(* IEC 61131-3 sources: AXOpen/src/showcase/app/src/core/AXOpen.Dialogs, 3 files *)

(* ---- AxoAlertDocuExample.st ---- *)
USING AXOpen.Core;

NAMESPACE AxoAlertExamples

    {S7.extern=ReadWrite}
    CLASS AxoAlertDocuExample EXTENDS AXOpen.Core.AxoObject
        //<AlertDeclaration>
        VAR PUBLIC
            {#ix-set:AttributeName = "<#Process Alert#>"}
            _alert : AXOpen.Core.AxoAlert;
        END_VAR
        //</AlertDeclaration>

        //<AlertUsageVariables>
        VAR PUBLIC
            {#ix-set:AttributeName = "<#Trigger alert#>"}
            _triggerAlert : BOOL;
            {#ix-set:AttributeName = "<#Alert was shown#>"}
            _alertWasShown : BOOL;
        END_VAR
        //</AlertUsageVariables>

        METHOD PUBLIC Execute
            //<AlertShowPattern>
            // AxoAlert shows a timed notification banner on the HMI.
            // Unlike AxoDialog, it does NOT wait for user response.
            // IsShown() returns TRUE once the alert has been displayed and dismissed.
            IF _triggerAlert THEN
                IF _alert.Show(THIS)
                    .WithTitle('<#Process Notification#>')
                    .WithType(eDialogType#Info)
                    .WithMessage('<#Cycle completed successfully.#>')
                    .WithTimeToBurn(UINT#5).IsShown() THEN
                    // Alert was displayed and timed out
                    _alertWasShown := TRUE;
                    _triggerAlert := FALSE;
                END_IF;
            END_IF;
            //</AlertShowPattern>
        END_METHOD

        METHOD AlertTypeExamples
        //<AlertTypes>
            // Info alert — general information
            IF _alert.Show(THIS)
                .WithTitle('<#Info#>')
                .WithType(eDialogType#Info)
                .WithMessage('<#Operation started.#>')
                .WithTimeToBurn(UINT#3).IsShown() THEN
                ;
            END_IF;

            // Success alert — operation completed
            IF _alert.Show(THIS)
                .WithTitle('<#Success#>')
                .WithType(eDialogType#Success)
                .WithMessage('<#Part inspection passed.#>')
                .WithTimeToBurn(UINT#5).IsShown() THEN
                ;
            END_IF;

            // Warning alert — attention needed
            IF _alert.Show(THIS)
                .WithTitle('<#Warning#>')
                .WithType(eDialogType#Warning)
                .WithMessage('<#Approaching maintenance interval.#>')
                .WithTimeToBurn(UINT#8).IsShown() THEN
                ;
            END_IF;

            // Danger alert — critical condition
            IF _alert.Show(THIS)
                .WithTitle('<#Danger#>')
                .WithType(eDialogType#Danger)
                .WithMessage('<#Emergency stop triggered.#>')
                .WithTimeToBurn(UINT#10).IsShown() THEN
                ;
            END_IF;
        //</AlertTypes>

        //<AlertRestore>
            // Restore clears the alert state, allowing it to be shown again
            _alert.Restore();
        //</AlertRestore>
        END_METHOD
    END_CLASS
END_NAMESPACE

(* ---- AxoDialogExamples.st ---- *)
USING AXOpen.Core;

NAMESPACE AxoDialogExamples

    {S7.extern=ReadWrite}
    CLASS Dialogs EXTENDS AXOpen.Core.AxoObject
        //<DialogDeclaration>
        VAR PUBLIC

            {#ix-set:AttributeName = "Restore All"}
            _invokeRestoreAll : BOOL;

            {#ix-set:AttributeName = "Call ALL"}
            _invokeCallAll : BOOL;

            {#ix-set:AttributeName = "Call ALL in Sequnce"}
            _invokeSequnceAll : BOOL;

             {#ix-set:AttributeName = "Dialog AA"}
             AA : AxoDialogTest;

             {#ix-set:AttributeName = "Dialog BB"}
             BB : AxoDialogTest;

             init_done : bool := false;
        END_VAR
        //</DialogDeclaration>
        VAR PRIVATE
            _rootObject : AxoObject;
        END_VAR

        METHOD PUBLIC Execute
            //<DialogExecution>
            if not init_done THEN
                AA.Caption := 'AA caption';
                BB.Caption := 'BB caption';

                AA.Question := 'AA Question';
                BB.Question := 'BB Question';

                init_done := true;
            end_if;

            IF _invokeRestoreAll THEN
                AA._restoreDialog := TRUE;
                BB._restoreDialog := TRUE;
                _invokeRestoreAll := FALSE;
            END_IF;

            IF _invokeCallAll THEN
                AA._callDialog := TRUE;
                BB._callDialog := TRUE;
                _invokeCallAll := FALSE;
            END_IF;

            IF _invokeSequnceAll THEN
                AA._callDialogInSequnce := TRUE;
                BB._callDialogInSequnce := TRUE;
                _invokeSequnceAll := FALSE;
            END_IF;

            _rootObject.Run(THIS);
            AA.Run(_rootObject);
            BB.Run(_rootObject);
            //</DialogExecution>
        END_METHOD
    END_CLASS
END_NAMESPACE

(* ---- AxoDialogTest.st ---- *)
USING AXOpen.Core;

NAMESPACE AxoDialogExamples

    {S7.extern=ReadWrite}
    CLASS AxoDialogTest EXTENDS AxoObject
        VAR PUBLIC

            {#ix-set:AttributeName = "Restore dialog"}
            _restoreDialog : BOOL;

            {#ix-set:AttributeName = "Call dialog"}
            _callDialog : BOOL;

            {#ix-set:AttributeName = "Call dialog in sequnce"}
            _callDialogInSequnce : BOOL;
            {#ix-set:AttributeName = "Iteration"}
            _iterationStep : INT;
            _timeOutCounter : INT;

            {#ix-set:AttributeName = "Generate Alerts in sequnce"}
            _alertInSequnce : BOOL;
            _alertIterationStep : INT;

            {#ix-set:AttributeName = "External Button signal - OK"}
            _externButtonSignal_ok : BOOL;
            {#ix-set:AttributeName = "External Button signal - YES"}
            _externButtonSignal_yes : BOOL;
            {#ix-set:AttributeName = "External Button signal - NO"}
            _externButtonSignal_no : BOOL;
            {#ix-set:AttributeName = "External Button signal - CANCEL"}
            _externButtonSignal_cancel : BOOL;

            Caption : STRING := 'Caption';
            Question : STRING := 'Question';

            {#ix-set:AttributeName = "Dialog Answer"}
            _answer : eDialogAnswer;

            {#ix-set:AttributeName = "Dialog"}
            _dialog : AXOpen.Core.AxoDialog;

            {#ix-set:AttributeName = "Alert Dialog"}
            _alertDialog : AXOpen.Core.AxoAlert;
        END_VAR

        METHOD PUBLIC OVERRIDE Run
            VAR_INPUT
                inParent : IAxoObject;
            END_VAR;

            SUPER.Run(inParent);
            // THIS.InitializeWithContext(_context);

            IF(_restoreDialog) THEN
                _restoreDialog := false;
                _dialog.Restore();
                _alertDialog.Restore();
                _callDialog:= false;
                _callDialogInSequnce := false;
                _iterationStep := 0;
                _timeOutCounter := 0;

                _alertInSequnce := FALSE;
                _alertIterationStep := 0;
            END_IF;

            //<DialogShowSimplePattern>
            //----------------------  SIMPLE DIALOG (HMI-only response) -------
            IF(_callDialog) THEN
               _answer := _dialog.Show(THIS)
                                  .WithCaption(Caption)
                                  .WithText(Question)
                                  .WithYesNoCancel()
                                  .WithType(eDialogType#Warning)
                                  .Answer();

                IF _answer <> eDialogAnswer#NoAnswer THEN
                    _callDialog := FALSE;
                END_IF;
            END_IF;
            //</DialogShowSimplePattern>

            //<DialogShowWithExternalClosePattern>
            //----------------------  DIALOG WITH EXTERNAL CLOSE SIGNALS -------
            IF(_callDialog) THEN
               _answer := _dialog.ShowWithExternalClose(THIS, _externButtonSignal_ok, _externButtonSignal_yes, _externButtonSignal_no, _externButtonSignal_cancel)
                                                .WithYesNoCancel()
                                                .WithType(eDialogType#Warning)
                                                .WithCaption(Caption)
                                                .WithText(Question)
                                                .Answer();

                IF _answer <> eDialogAnswer#NoAnswer THEN
                    _callDialog := FALSE;
                END_IF;
            END_IF;
            //</DialogShowWithExternalClosePattern>

            //<DialogSequencePattern>
            //----------------------  DIALOG IN SEQUNCE-------------------
            IF _callDialogInSequnce THEN

                if  _iterationStep  = 0 then
                    _iterationStep := _iterationStep + 1;
                end_if;

                if  _iterationStep  = 1 then

                    if not _dialog.HasError() then
                        _answer := _dialog.ShowWithExternalClose(THIS, _externButtonSignal_ok, _externButtonSignal_yes, _externButtonSignal_no, _externButtonSignal_cancel)
                        .WithYesNoCancel()
                        .WithType(eDialogType#Info)
                        .WithCaption( 'Iteraion 1')
                        .WithText(Question)
                        .Answer();

                        THIS.Watcher_Monitor();
                        if _answer <> eDialogAnswer#NoAnswer THEN
                            THIS.Watcher_Reset();
                            _iterationStep := _iterationStep + 1;
                        END_IF;

                    end_if;

                end_if;

                if  _iterationStep  = 2 then

                    if not _dialog.HasError() then
                        _answer := _dialog.ShowWithExternalClose(THIS, _externButtonSignal_ok, _externButtonSignal_yes, _externButtonSignal_no, _externButtonSignal_cancel)
                        .WithYesNoCancel()
                        .WithType(eDialogType#Success)
                        .WithCaption('Iteraion 2')
                        .WithText(Question)
                        .Answer();

                        THIS.Watcher_Monitor();
                        if _answer <> eDialogAnswer#NoAnswer THEN
                            THIS.Watcher_Reset();
                            _iterationStep := _iterationStep + 1;
                        END_IF;
                    end_if;

                end_if;

                if  _iterationStep  = 3 then
                    if not _dialog.HasError() then
                        _answer := _dialog.ShowWithExternalClose(THIS, _externButtonSignal_ok, _externButtonSignal_yes, _externButtonSignal_no, _externButtonSignal_cancel)
                        .WithYesNoCancel()
                        .WithType(eDialogType#Warning)
                        .WithCaption('Iteraion 3')
                        .WithText(Question)
                        .Answer();

                        THIS.Watcher_Monitor();
                        if _answer <> eDialogAnswer#NoAnswer THEN
                            THIS.Watcher_Reset();
                            _iterationStep := _iterationStep + 1;
                        END_IF;
                    end_if;

                end_if;

                if  _iterationStep  = 4 then
                    if not _dialog.HasError() then
                        _answer := _dialog.ShowWithExternalClose(THIS, _externButtonSignal_ok, _externButtonSignal_yes, _externButtonSignal_no, _externButtonSignal_cancel)
                        .WithYesNoCancel()
                        .WithType(eDialogType#Danger)
                        .WithCaption('Iteraion 4')
                        .WithText(Question)
                        .Answer();

                        THIS.Watcher_Monitor();
                        if _answer <> eDialogAnswer#NoAnswer THEN
                            THIS.Watcher_Reset();
                            _iterationStep := _iterationStep + 1;
                        END_IF;
                    end_if;

                end_if;

            end_if;
            //</DialogSequencePattern>
            //<AlertDialogPattern>
            //---------------------- ALERT DIALOG -------------------
            IF _alertInSequnce THEN

                if  _alertIterationStep  = 0 then
                    _alertIterationStep := _alertIterationStep + 1;
                end_if;

                if  _alertIterationStep  = 1 then
                    if not _alertDialog.HasError() then
                        IF _alertDialog.Show(THIS)
                            .WithTitle(Caption)
                            .WithType(eDialogType#Info)
                            .WithMessage('Alert stage 1!')
                            .WithTimeToBurn(UINT#5).IsShown()  THEN
                            //when task is done, move next
                            _alertIterationStep := _alertIterationStep + 1;
                        END_IF;
                    end_if;
                end_if;

                if  _alertIterationStep  = 2 then
                    if not _alertDialog.HasError() then
                        IF _alertDialog.Show(THIS)
                            .WithTitle(Caption)
                            .WithType(eDialogType#Success)
                            .WithMessage('Alert stage 2!')
                            .WithTimeToBurn(UINT#5).IsShown() THEN
                            //when task is done, move next
                            _alertIterationStep := _alertIterationStep + 1;
                        END_IF;
                    end_if;
                end_if;

                if  _alertIterationStep  = 3 then
                    if not _alertDialog.HasError() then
                        IF _alertDialog.Show(THIS)
                            .WithTitle(Caption)
                            .WithType(eDialogType#Warning)
                            .WithMessage('Alert stage 3')
                            .WithTimeToBurn(UINT#5).IsShown() THEN
                            //when task is done, move next
                            _alertIterationStep := _alertIterationStep + 1;
                        END_IF;
                    end_if;
                end_if;

                if  _alertIterationStep  = 4 then
                    if not _alertDialog.HasError() then
                        IF _alertDialog.Show(THIS)
                            .WithTitle(Caption)
                            .WithType(eDialogType#Danger)
                            .WithMessage('Alert stage 4')
                            .WithTimeToBurn(UINT#5).IsShown() THEN
                            //when task is done, move next
                            _alertIterationStep := _alertIterationStep + 1;
                        END_IF;
                    end_if;
                end_if;

                if  _alertIterationStep  = 5 then
                    if not _alertDialog.HasError() then
                        IF _alertDialog.Show(THIS)
                            .WithTitle(Caption)
                            .WithType(eDialogType#Undefined)
                            .WithMessage('Alert stage 5')
                            .WithTimeToBurn(UINT#5).IsShown()  THEN
                            //when task is done, move next
                            _alertIterationStep := _alertIterationStep + 1;
                        END_IF;
                    end_if;
                end_if;

                if  _alertIterationStep  >= 6 then  // simulate time gap
                    _alertIterationStep := 0 ;
                end_if;

            ELSE
                _alertIterationStep := 0 ;
                if _alertDialog.HasError() THEN
                    _alertDialog.Restore();
                END_IF;

            END_IF;
            //</AlertDialogPattern>
        END_METHOD

        METHOD PRIVATE Watcher_Monitor
            _timeOutCounter := _timeOutCounter + 1;
            if _timeOutCounter > 300 then
                _externButtonSignal_cancel := true;
            END_IF;
        END_METHOD

        METHOD PRIVATE Watcher_Reset
            _timeOutCounter := 0;
            _externButtonSignal_cancel := false;
            _externButtonSignal_ok := false;
            _externButtonSignal_yes := false;
            _externButtonSignal_no := false;
        END_METHOD

    END_CLASS
END_NAMESPACE
